{attribute 'linkalways'} 
{attribute 'no_explicit_call' := 'This FB is a CLASS and must be accessed using methods or properties'}
{attribute 'enable_dynamic_creation'}
FUNCTION_BLOCK FINAL EQ_WORD EXTENDS Node
VAR
	in1 : _WORD(0);
	in2 : _WORD(0);
	out : _BOOL(FALSE);
END_VAR

METHOD PUBLIC Clone : I_Node
VAR
	pNode : POINTER TO EQ_WORD;
END_VAR
pNode := __NEW(EQ_WORD);
Clone := pNode^;
END_METHOD

METHOD FB_init : BOOL
VAR_INPUT
	bInitRetains : BOOL; // if TRUE, the retain variables are initialized (warm start / cold start)
	bInCopyCode : BOOL;  // if TRUE, the instance afterwards gets moved into the copy code (online change)
END_VAR
AddInput('in1',THIS^.in1);
AddInput('in2',THIS^.in2);
AddOutput('out', THIS^.out);
END_METHOD

METHOD PROTECTED OnExecute
VAR
END_VAR
out.Value := in1.Value = in2.Value;
END_METHOD

END_FUNCTION_BLOCK

(* stored: Version 1.1.0.1, ProductVersion 3.1.4024.15
   POU EQ_WORD: Id {c5127fb0-3074-4b0c-8662-a3784dafb59a}, SpecialFunc None
   Folder Constructor: Id {62f4dd6a-b54a-4ae0-8381-3d57a7894b9d}
   Method Clone: Id {78b02c6c-c65a-45b0-a237-ff7c3aebdc58}
   Method FB_init: Id {0290e11c-2a4f-45fd-8178-095424e9a011}
   Method OnExecute: Id {c651d354-8516-4329-bce4-733f0fe7ce26} *)
